(* Reads the NC axis parameter set for the owning axis and reports completion
   through I_Initializable.

   Unlike Mc3AxisParameterLoader this has no parameter table: MC_ReadParameterSet
   fetches the whole ST_AxisParameterSet in one call, so there is nothing to
   enumerate. The owning axis picks the fields it needs off AxisParameterSet.
   Call Configure() once with the axis reference, then Initialize() cyclically
   until Initialized or Error. *)
FUNCTION_BLOCK Mc2AxisParameterLoader IMPLEMENTS I_Initializable
VAR
	_Axis			   : REFERENCE TO Tc2_MC2.AXIS_REF;
	_AxisParameters	   : Tc2_MC2.ST_AxisParameterSet;
	_Initialized	   : BOOL;
	_Error			   : BOOL;
	MCReadParameterSet : Tc2_MC2.MC_ReadParameterSet;
END_VAR

(* The parameter set as read from the NC. Only meaningful once Initialized. *)
PROPERTY AxisParameterSet : REFERENCE TO Tc2_MC2.ST_AxisParameterSet
GET
AxisParameterSet REF= _AxisParameters;
END_GET
END_PROPERTY

(* Binds the loader to the NC axis it should read from. *)
METHOD Configure
VAR_INPUT
	Axis : REFERENCE TO Tc2_MC2.AXIS_REF;
END_VAR
_Axis REF= Axis;
END_METHOD

{attribute 'monitoring' := 'call'}
PROPERTY Error : BOOL
GET
Error := _Error;
END_GET
END_PROPERTY

METHOD Initialize
IF _Initialized OR _Error THEN
	RETURN;
END_IF

IF NOT __ISVALIDREF(_Axis) THEN
	RETURN;
END_IF

MCReadParameterSet(Parameter := _AxisParameters, Axis := _Axis, Execute := TRUE);

IF MCReadParameterSet.Busy THEN
	RETURN;
END_IF

IF MCReadParameterSet.Error THEN
	_Error := TRUE;
ELSIF MCReadParameterSet.Done THEN
	_Initialized := TRUE;
END_IF

MCReadParameterSet(Parameter := _AxisParameters, Axis := _Axis, Execute := FALSE);
END_METHOD

{attribute 'monitoring' := 'call'}
PROPERTY Initialized : BOOL
GET
Initialized := _Initialized;
END_GET
SET
_Initialized := Initialized;

// Clearing the flag restarts the read
IF NOT Initialized THEN
	_Error := FALSE;
	MCReadParameterSet(Parameter := _AxisParameters, Axis := _Axis, Execute := FALSE);
END_IF
END_SET
END_PROPERTY

END_FUNCTION_BLOCK

(* stored: Version 1.1.0.1, ProductVersion 3.1.4026.20
   POU Mc2AxisParameterLoader: Id {daa43417-7960-4f86-8309-739dd27116f0}, SpecialFunc None
   Property AxisParameterSet: Id {e076ed6d-a824-4d9a-8c49-deb2e2b4b2c7}
   Get Get: Id {bb81b6f9-374e-4f10-a430-5b01e455c93f}
   Method Configure: Id {a4acdc71-ec24-43fc-a075-d187cd28f20e}
   Property Error: Id {4a9b1614-d1ae-42c5-904a-1f6a61e6586b}
   Get Get: Id {1c808876-14d5-4b6d-9374-c8e16891960f}
   Method Initialize: Id {09a31372-7751-4d69-9a4f-08fb3fe65391}
   Property Initialized: Id {397ef0f0-64ff-4203-8cda-1e72e5fb6492}
   Get Get: Id {6c063041-7fa5-48d5-9f5e-557a98b25826}
   Set Set: Id {29b55b76-9669-4d72-b3bd-dc12f7de8a34} *)
